// TIA Portal V19 export
FUNCTION_BLOCK "TYPIC_C302_BF_LKM"   // FB68, FBD
TITLE = TYPIC_C302_BF_LKM: Luchtkwaliteitsmeting verkeerskoker
{ S7_Optimized_Access := 'TRUE' }
AUTHOR : OCOTECH
FAMILY : Typical
NAME : C302.801
// Logisch Object Besturing: C302.801
// 
// Het doel van de luchtkwaliteitsmeting is het meten van de zichtcondities in de verkeerskoker om op basis daarvan een indicatie te krijgen van de luchtkwaliteit in de verkeerskoker en rook in de verkeerskoker te detecteren.
// stored: MemoryReserve 10, SetENOAutomatically false
   VAR_INPUT
      STU_ALG_LCK_SIG { ExternalAccessible := 'False'; ExternalVisible := 'False'; ExternalWritable := 'False'} : USInt;   // Onderdruk alarmen
      CFG_SWA1 { ExternalAccessible := 'False'; ExternalVisible := 'False'; ExternalWritable := 'False'} : Real;   // Grenswaarde waarboven aangenomen wordt dat er lichte zichtbeperking is
      CFG_SWA2 { ExternalAccessible := 'False'; ExternalVisible := 'False'; ExternalWritable := 'False'} : Real;   // Grenswaarde waarboven aangenomen wordt dat er matige zichtbeperking is
      CFG_SWA3 { ExternalAccessible := 'False'; ExternalVisible := 'False'; ExternalWritable := 'False'} : Real;   // Grenswaarde waarboven aangenomen wordt dat er waarneembare zichtbeperking is
      CFG_SWA4 { ExternalAccessible := 'False'; ExternalVisible := 'False'; ExternalWritable := 'False'} : Real;   // Grenswaarde waarboven aangenomen wordt dat er ernstige zichtbeperking is
      CFG_HYS { ExternalAccessible := 'False'; ExternalVisible := 'False'; ExternalWritable := 'False'} : Real;   // Hysteresis om naar lagere aanduiding te gaan voor zichtkwaliteit
      CFG_MAX_NOK { ExternalAccessible := 'False'; ExternalVisible := 'False'; ExternalWritable := 'False'} : Int;   // Aantal opeenvolgende niet observeerbare luchtkwaliteitsmeters voor beschikbaarheidsstatus beperkt beschikbaar
   END_VAR
   VAR_OUTPUT
      VAR_ROOK { ExternalAccessible := 'False'; ExternalVisible := 'False'; ExternalWritable := 'False'} : USInt;   // Rookdetectie
      VAR_POS_ROOK { ExternalAccessible := 'False'; ExternalVisible := 'False'; ExternalWritable := 'False'} : Bool;   // Positie van de rookdetectie
      VAR_LKM_BWA { ExternalAccessible := 'False'; ExternalVisible := 'False'; ExternalWritable := 'False'} : Real;   // Meetwaarde luchtkwaliteit (maximumwaarde in koker)
   END_VAR
   VAR_IN_OUT
      VAR_LKM : Array[0..1] of Bool;   // Array met alle luchtkwaliteitsmeters, met alle variabelen van de luchtkwaliteitsmeter
   END_VAR
   VAR
      SIG { ExternalWritable := 'False'} : Struct   // Signaleringen
         AA01 : Bool;   // Openvolgende luchtkwaliteitsmeters niet observeerbaar
         AB01 : Bool;   // Luchtkwaliteitsmeting niet beschikbaar
         AB02 : Bool;   // Luchtkwaliteitsmeting beperkt beschikbaar
         AV01 : Bool;   // Rook gedetecteerd
         AV02 : Bool;   // Slecht zicht gedetecteerd
      END_STRUCT;
      VAR { ExternalWritable := 'False'} : Struct   // Variabelen
         BSC : USInt;   // Geeft de beschikbaarheid aan van de luchtkwaliteitsmeting aan
         VGV_SIG_VOP : Bool;   // TRUE = Signaleringen vrijgegeven voor verkeersoperator FALSE = Onderdrukt
         STS_BWA : USInt;   // Indicatie van de zichtbeperking (zichtconditie) in de tunnel
         POS { ExternalAccessible := 'False'; ExternalVisible := 'False'} : USInt;   // Positie in de tunnel van luchtkwaliteitsmeter die hoogste geldige k-waarde aangeeft
         "2oo3_BWA" { ExternalAccessible := 'False'; ExternalVisible := 'False'} : USInt;   // k-waarde als resultaat van 2oo3 filter
         "2oo3_POS" { ExternalAccessible := 'False'; ExternalVisible := 'False'} : USInt;   // Positie met hoogste k-waarde vanuit 2oo3 filter
         "2oo3_GEM" { ExternalAccessible := 'False'; ExternalVisible := 'False'} : USInt;   // Gemiddelde van de 3-metingen bij 2oo3 filter
         "2oo3_HULP1" { ExternalAccessible := 'False'; ExternalVisible := 'False'} : USInt;   // Gemiddelde van meting 2 en 3
         "2oo3_HULP2" { ExternalAccessible := 'False'; ExternalVisible := 'False'} : USInt;   // Gemiddelde van meting 1 en 3
         "2oo3_HULP3" { ExternalAccessible := 'False'; ExternalVisible := 'False'} : USInt;   // Gemiddelde van meting 1 en 2
         "2oo3_HULP4" { ExternalAccessible := 'False'; ExternalVisible := 'False'} : USInt;   // Procentuele afwijking HULP1 met GEM
         "2oo3_HULP5" { ExternalAccessible := 'False'; ExternalVisible := 'False'} : USInt;   // Procentuele afwijking HULP2 met GEM
         "2oo3_HULP6" { ExternalAccessible := 'False'; ExternalVisible := 'False'} : USInt;   // Procentuele afwijking HULP3 met GEM
         LKM_HULP { ExternalAccessible := 'False'; ExternalVisible := 'False'} : USInt;   // Hulpvariabele voor tussenresultaten
      END_STRUCT;
   END_VAR
BEGIN

REGION Network 1: START
END_REGION

REGION Network 2: +++ Bepalen meetwaarde luchtkwaliteitsmeting +++
   // Éen algemene meetwaarde voor de verkeerskoker bepalen op basis van de individuele metingen van alle luchtkwaliteitsmeters waarbij defecte luchtkwaliteitsmeters en afwijkende meetwaardes er uit gefilterd worden
END_REGION

REGION Network 3: +++ Indicatie zichtcondities +++
   // Zichtconditie in de verkeerskoker bepalen (Geen zichtbeperking / Lichte zichtbeperking / Matige zichtbeperking / Waarneembare zichtbeperking / Ernstige zichtbeperking).
END_REGION

REGION Network 4: +++ Rookdetectie +++
   // Aangeven van rookdetectie in de verkeerskoker en de lengtepositie in de verkeerskoker van de rookdetectie.
END_REGION

REGION Network 5: +++ Bepalen beschikbaarheidsstatus +++
   // Beschikbaarheidsstatus (beschikbaar / beperkt beschikbaar / niet beschikbaar) bepalen.
END_REGION

REGION Network 6 (SCL): Beschikbaarheidsstatus bepalen
   IF 
       //voorwaarden "Niet beschikbaar"
       TRUE
   THEN
       //Beschikbaarheidsstatus = Niet Beschikbaar
       #VAR.BSC:= "NietBeschikbaar";
   ELSIF
       //voorwaarden "Beperkt beschikbaar"
       TRUE
   THEN
       //Beschikbaarheidsstatus = Beperkt Beschikbaar
       #VAR.BSC:= "Beperkt";
   ELSE
       //Beschikbaarheidsstatus = Beschikbaar
       #VAR.BSC:= "Beschikbaar";
   END_IF;
END_REGION

REGION Network 7: +++ Signaleringen +++
   // Aanmaken signaleringen.
END_REGION

REGION Network 8: Signalering AB01 : Niet Beschikbaar
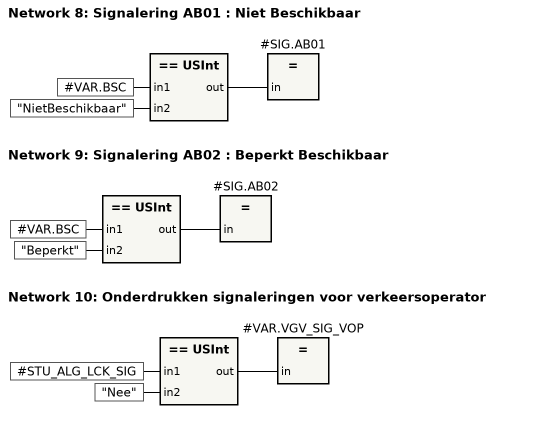
   #SIG.AB01 := #VAR.BSC = "NietBeschikbaar";
END_REGION

REGION Network 9: Signalering AB02 : Beperkt Beschikbaar
   #SIG.AB02 := #VAR.BSC = "Beperkt";
END_REGION

REGION Network 10: Onderdrukken signaleringen voor verkeersoperator
   // Via de variabele VGV_SIG_VOP wordt aan IRIS SCADA doorgegeven of signaleringen (bestemd voor de verkeersoperator) van de deze functie zichtbaar (of onderdrukt) moeten zijn.
   #VAR.VGV_SIG_VOP := #STU_ALG_LCK_SIG = "Nee";
END_REGION

REGION Network 11: EINDE
   // Variabelen van intern scada rakvlak naar outputs copieren
END_REGION
END_FUNCTION_BLOCK
